SUBAPPLICATION logiBUS_PI_Raw_Publish_OPC (* logiBUS_PI_IDA (Puls-Eingang) rein als Frequenz (Hz, REAL) lesen + per OPC-UA publizieren, OHNE jegliche VT-Interaktion und ohne Kanal-Enable/Status. Fuer Geschwindigkeitssensoren (Impulsgeber), deren physischer Puls-Eingang auf einer Station OHNE VT-Anschluss sitzt (z.B. Aufnahmegeschwindigkeit B03, Igelband B10/B11 auf APIXON STG2/STG3) - die km/h-Umrechnung + VT-Anzeige laufen dann auf der Station mit VT-Anschluss, gespeist per Remote-Subscribe dieser Frequenz (analog zu logiBUS_AI_Raw_Publish_OPC / logiBUS_AI_Calibrate_Remote_IDA_OPC). *)
  (* Standard: 61499-2; Description: Copyright (c) 2026 Meisterschulen am Ostbahnhof This program and the accompanying materials are made available under the terms of the Eclipse Public License 2.0 which is available at https://www.eclipse.org/legal/epl-2.0/ SPDX-License-Identifier: EPL-2.0 *)
  (* Version 1.0, 2026-09-12, Franz Höpfinger, Meisterschulen am Ostbahnhof, initial implementation - schlanke Frequenz-Rohwert-Haelfte von logiBUS_PI_IDA_OPC (ohne Kanal-Enable/VT-Status/Zaehler-Publish), fuer Sensoren auf einer Station ohne VT-Anschluss (B03/B10/B11). *)
  (* Version 1.3, 2026-10-03, Franz Höpfinger, Meisterschulen am Ostbahnhof, Folgefix zu FT_DERIV_10_AR v1.2 (K jetzt AUI-Adapter-Socket statt Parameter): bisheriges Parameter Name='K' Value='9' auf FT_DERIV_10_AR entfernt (waere jetzt ein IDE-Fehler, da K kein plain InputVar mehr ist), ersetzt durch LIT_DerivK (initval_AUI, INIT_VAL=9) + AdapterConnection auf FT_DERIV_10_AR.K - gleicher Wert wie bisher, nur adapter-konform verdrahtet. *)
  (* Version 1.2, 2026-10-03, Franz Höpfinger, Meisterschulen am Ostbahnhof, Franz (Zapfwelle B21 auf STG4): 'soll VORHER auf dieselbe Einheit gerundet werden wie RPTO, 0.125 U/min, genauer muss es nicht sein' - neuer OSCAT_adapter::Mathematical::ROUND_STEP_AR zwischen FT_PT1_AR und AR_PUBLISH_HZ eingefuegt, neuer InputVar RASTER_HZ (Default 0.0001 Hz = praktisch kein Runden, fuer bestehende Aufrufer Aufnahme B03/Igelband B10/B11 unveraendert) - Zapfwelle setzt per Parameter RASTER_HZ=0.00208333 (= 0.125 U/min / 60 Hz->U/min-Faktor). *)
  (* Version 1.1, 2026-09-22, Franz Höpfinger, Meisterschulen am Ostbahnhof, PT1-Filterzeit einstellbar + INI-persistiert statt hartcodiertem T#2s-Literal (initval_ATM entfernt) - Franz: 'Kunde will die Filter Zeit ohnehin Einstellbar haben (die 2S), Abspeichern in INI, 2S als Standardwert'. Neue FilterTimeS (NumericValue_TO_AR2_OPC, Sekunden REAL, VT+Web mergebar) + INI_FilterTimeS (INI_AR2, Section/Key='FilterTimeS', Default REAL#2.0) + neuer Baustein AR_S_TO_ATM (Sekunden-REAL -> TIME, x1000 + numerische Konvertierung) speisen FT_PT1_AR.TM. FT_PT1_AR.INIT wird jetzt von INI_FilterTimeS.INITO ausgeloest (statt initval_ATM.INITO) - ein Wert, der zur Laufzeit per VT/Web geaendert wird, greift damit erst nach einem Neustart der Station (bewusste Vereinfachung, kein Live-Re-Init um Filter-Transienten waehrend des Betriebs zu vermeiden). Neue InputVars stObjFilterTimeS/ID_FILTER_TIME_READ/ID_FILTER_TIME_WRITE/sSection - bestehende Aufrufer muessen diese nachziehen (siehe Inputs_STG2/STG3.SUB), sonst laufen AR_SUBSCRIBE_1/AR_PUBLISH_1/INI_AR2 mit leeren IDs. *)
  PACKAGE MyLib::sys;
  IMPORT logiBUS::io::PI::logiBUS_PI;
  IMPORT logiBUS::io::PI::logiBUS_PI_S;
  IMPORT isobus::UT::Q::const::IDs::ID_NULL;
  IMPORT logiBUS::utils::conversion::phys::NumericObjectPool_S;
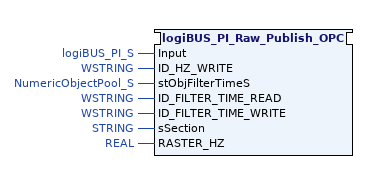
  VAR_INPUT
    Input : logiBUS::io::PI::logiBUS_PI_S := logiBUS_PI::Invalid; (* Identify the Input PulseInput_I1..I9 *)
    ID_HZ_WRITE : WSTRING; (* Frequenz-Publish-Adresse (REAL Hz, ACTION=PUBLISH), lokal auf dieser Station *)
    stObjFilterTimeS : logiBUS::utils::conversion::phys::NumericObjectPool_S := (u16ObjId := ID_NULL, r32Scale := 1.0, i32Offset := 0, u8Decimals := 1); (* Object ID + Scale/Offset/Decimals CNumberVariable (PT1-Filterzeit in Sekunden, VT-Eingabefeld) *)
    ID_FILTER_TIME_READ : WSTRING; (* Remote-Subscribe-Adresse (REAL Sekunden, ACTION=SUBSCRIBE) fuer Web-Override der Filterzeit *)
    ID_FILTER_TIME_WRITE : WSTRING; (* Lokale Echo/Re-Publish-Adresse (REAL Sekunden, ACTION=PUBLISH) der aktuellen Filterzeit *)
    sSection : STRING; (* INI settings.ini Section fuer die persistierte Filterzeit (eindeutig pro Sensor-Instanz) *)
    RASTER_HZ : REAL := 0.0001; (* Rundungsraster (Hz) vor AR_PUBLISH_HZ - Platzhalter-Default 0.0001 (praktisch kein Runden, fuer bestehende Aufrufer unveraendert), per Parameter auf die gewuenschte Aufloesung setzen (z.B. 0.00208333 = 0.125 U/min bei SCALE=60 Hz->U/min stromabwaerts) *)
  END_VAR
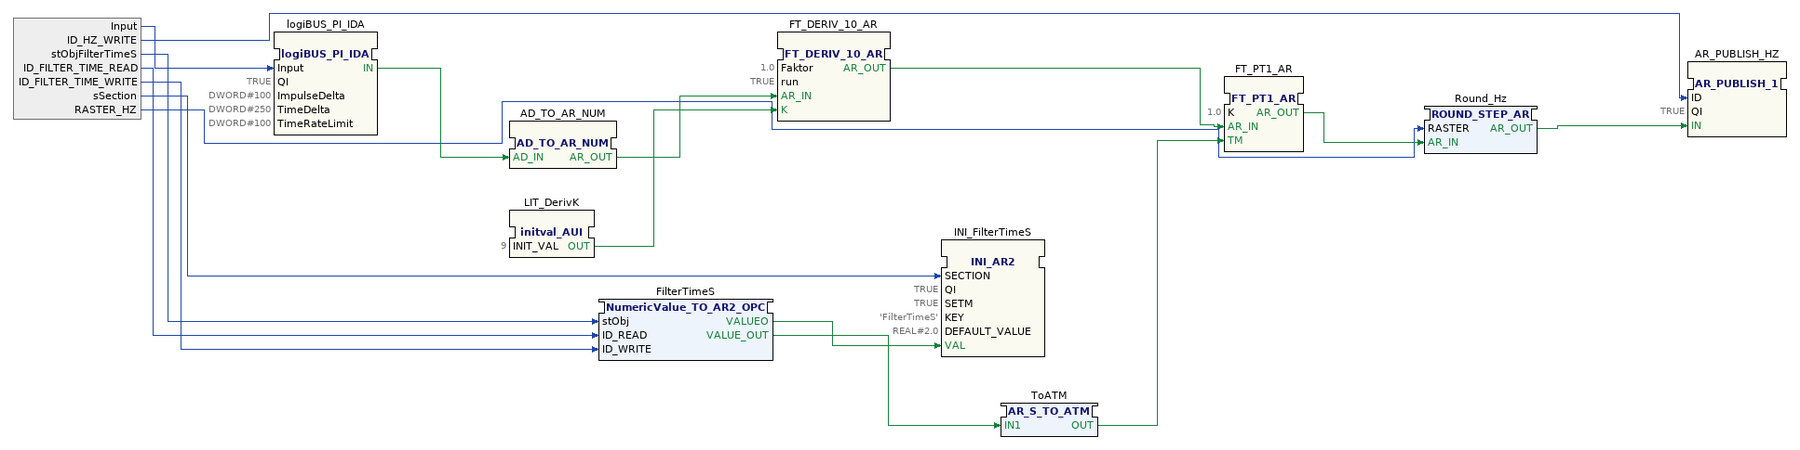
  FBS
    logiBUS_PI_IDA : logiBUS::io::PI::logiBUS_PI_IDA(QI := TRUE, ImpulseDelta := DWORD#100, TimeDelta := DWORD#250, TimeRateLimit := DWORD#100);
    AD_TO_AR_NUM : adapter::conversion::unidirectional::AD_TO_AR_NUM;
    FT_DERIV_10_AR : OSCAT_adapter::Control::FT_DERIV_10_AR(Faktor := 1.0, run := TRUE);
    LIT_DerivK : adapter::types::unidirectional::AUI::initval::initval_AUI(INIT_VAL := 9);
    FT_PT1_AR : OSCAT_adapter::Control::FT_PT1_AR(K := 1.0);
    AR_PUBLISH_HZ : adapter::net::AR_PUBLISH_1(QI := TRUE);
    INI_FilterTimeS : eclipse4diac::storage::INI_AR2(QI := TRUE, SETM := TRUE, KEY := 'FilterTimeS', DEFAULT_VALUE := REAL#2.0);
  END_FBS
  SUBAPPS
    Round_Hz : OSCAT_adapter::Mathematical::ROUND_STEP_AR;
    FilterTimeS : MyLib::sys::NumericValue_TO_AR2_OPC;
    ToATM : MyLib::sys::AR_S_TO_ATM;
  END_SUBAPPS
  DATA_CONNECTIONS
    Input TO logiBUS_PI_IDA.Input;
    ID_HZ_WRITE TO AR_PUBLISH_HZ.ID;
    stObjFilterTimeS TO FilterTimeS.stObj;
    ID_FILTER_TIME_READ TO FilterTimeS.ID_READ;
    ID_FILTER_TIME_WRITE TO FilterTimeS.ID_WRITE;
    sSection TO INI_FilterTimeS.SECTION;
    RASTER_HZ TO Round_Hz.RASTER;
  END_CONNECTIONS
  ADAPTER_CONNECTIONS
    logiBUS_PI_IDA.IN TO AD_TO_AR_NUM.AD_IN;
    AD_TO_AR_NUM.AR_OUT TO FT_DERIV_10_AR.AR_IN;
    FT_DERIV_10_AR.AR_OUT TO FT_PT1_AR.AR_IN;
    LIT_DerivK.OUT TO FT_DERIV_10_AR.K;
    FilterTimeS.VALUEO TO INI_FilterTimeS.VAL;
    FilterTimeS.VALUE_OUT TO ToATM.IN1;
    ToATM.OUT TO FT_PT1_AR.TM;
    FT_PT1_AR.AR_OUT TO Round_Hz.AR_IN;
    Round_Hz.AR_OUT TO AR_PUBLISH_HZ.IN;
  END_CONNECTIONS
END_SUBAPPLICATION
